(* CoDeSys 2.3.9.47 project: pid_controller_1.pro *)
(* Libraries: STANDARD.LIB 5.6.98 11:03:02, C:\Users\Raphael\Documents\HSLU\05_HS_16\ATS\sharedFolder\Projects\Lab_4\lib_lab_4.lib 17.11.16 20:23:40 *)

(* Task configuration *)
TASK Standard (PRIORITY := 0, INTERVAL := T#10ms);
	MAIN
END_TASK

(* Global variable list: TwinCAT_Configuration *)
(* Generated automatically by TwinCAT - (read only) *)
VAR_CONFIG
	MAIN.mot_en AT %QX0.0 : BOOL;	(*  ~ {LinkedWith:TIID^Device 1 (EtherCAT)^Term 7 (EK1100)^Term 10 (EL7342)^DCM Control Channel 1^Control^Enable} *)
	MAIN.mot_v AT %QB4 : INT;	(*  ~ {LinkedWith:TIID^Device 1 (EtherCAT)^Term 7 (EK1100)^Term 10 (EL7342)^DCM Velocity Channel 1^Velocity} *)
	MAIN.cnt_OF AT %IX4.0 : BOOL;	(*  ~ {LinkedWith:TIID^Device 1 (EtherCAT)^Term 7 (EK1100)^Term 9 (EL5101)^ENC Status compact^Status^Counter overflow} *)
	MAIN.cnt_UF AT %IX4.1 : BOOL;	(*  ~ {LinkedWith:TIID^Device 1 (EtherCAT)^Term 7 (EK1100)^Term 9 (EL5101)^ENC Status compact^Status^Counter underflow} *)
	MAIN.cnt_val AT %IB8 : UINT;	(*  ~ {LinkedWith:TIID^Device 1 (EtherCAT)^Term 7 (EK1100)^Term 9 (EL5101)^ENC Status compact^Counter value} *)
END_VAR

(* Data type *)
TYPE PID_parameters :
STRUCT
(*Essential Parameters*)
Kp	:REAL;
Ti	:REAL;
Td	:REAL;
N	:REAL;
sat	:REAL;
(*Features*)
has_arw	:BOOL;
has_sat	:BOOL;
has_bra	:BOOL;

END_STRUCT
END_TYPE

(* POU MAIN, ST *)
PROGRAM MAIN
VAR
pid	: PID_Controller;
par	: PID_parameters;
ref	: REAL;
v_r : REAL;
out	: REAL;
(*Device Signals*)
mot_en	AT%Q*: BOOL;
mot_v	AT%Q*: INT;
cnt_OF	AT%I*: BOOL;
cnt_UF	AT%I*: BOOL;
cnt_val	AT%I*: UINT;
END_VAR
t_cycle := 0.01;
(*ref := SquareSignal(t_global, -1, 1);*)
v_r := 12;
ref := v_r*32768/24;

(*Essential Parameters*)
par.Kp	:= 1;
par.Ti	:= 0.1;
par.Td	:= 0.1;
par.N	:= 10;
par.sat	:= 100;
(*Features*)
par.has_arw	:= FALSE;
par.has_sat	:= FALSE;
par.has_bra	:= TRUE;


(*Initialize Controller*)
pid();
pid.r_k := ref;
out := pid.y_k;


(*Increment global Time*)
t_global := t_global + t_cycle;
END_PROGRAM

(* POU PID_Controller, ST *)
FUNCTION_BLOCK PID_Controller
VAR_INPUT
	r_k		: REAL;
	param	: PID_parameters;
END_VAR
VAR_OUTPUT
	y_k		: REAL;
END_VAR
VAR
	e_k		: REAL;
	e_k_1	: REAL;
	(*P-Part*)
	u_p_k	: REAL;
	(*I-Part*)
	u_i_k	: REAL;
	u_i_k_1	: REAL;
	(*D-Part*)
	u_d_k	: REAL;
	u_d_k_1	: REAL;
	a		: REAL;
	b		: REAL;
END_VAR
(*Calculate Error*)
e_k := r_k - y_k;
e_k := e_k * param.Kp;

a 	:= param.Td / (param.Td + param.N * t_cycle);
b	:= (param.Kp * param.Td * param.N)/(param.Td + param.N * t_cycle);

(*Proportional Term*)
u_p_k := e_k;

(*Integrator using Trapeze Approximation*)
u_i_k := u_i_k_1 + (e_k + e_k_1)*t_cycle/(2*param.Ti);

(*Derivate Term*)
IF (param.has_bra = TRUE) THEN
u_d_k := param.Kp * param.Td * (-y_k - e_k_1) / t_cycle;
ELSE
u_d_k := a*u_d_k_1 + b*(e_k - e_k_1);
END_IF

(*Calculate Output*)
PID_Controller.y_k := u_p_k + u_i_k + u_d_k;

(*Actualize later used Variables*)
e_k_1 	:= e_k;
u_i_k_1 := u_i_k;
u_d_k_1	:= u_d_k;
END_FUNCTION_BLOCK
